{attribute 'qualified_only'}
{attribute 'strict'}
TYPE E_Location :
(
	UNKNOWN := 0,
	INFEED,
	ALLIGNMENT,
//	PRE_DOCKING,
	DOCKING,
//	AIR_LOCK,
//	FLUSHING_CLEAN,
//	CLEAN_ROOM
);
END_TYPE

(* stored: Version 1.1.0.1, ProductVersion 3.1.4024.12
   DUT E_Location: Id {a212cb9f-20ff-4dea-8327-f50aeadd4b4d} *)
